Universal Robots PolyScope program: mt_rtde_control_loop_v4.urp

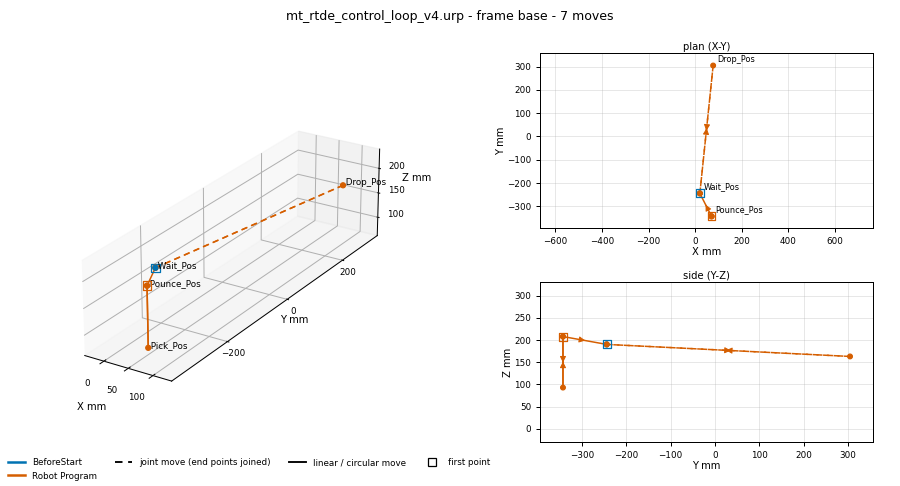
[picture p0: tool path of mt_rtde_control_loop_v4.urp in frame base, 7 of 7 moves have a stored position in this frame; points joined in program order, loops and branches not executed]
Program mt_rtde_control_loop_v4 (installation=mt_exhibit_v4 directory=/programs/usbdisk createdIn=3.2.19275.0 lastSavedIn=5.11.9.1010452 robotSerialNumber=20225300174)
Calibrated DH parameters: a=[-0.000135, -0.229339, -0.213305, 0.000029, -0.000076, 0]; d=[0.152122, 26.260282, -25.005713, -1.123774, 0.085381, 0.092263]; alpha=[1.57245, 0.003146, 0.006488, 1.570884, -1.571468, 0]; deltaTheta=[0, 0.345729, -0.307593, -0.038131, 0.000003, 0]
BeforeStart
  PRINTER_IDLE := 1
  PRINTER_RUNNING := 2
  COBOT_INIT := 0
  COBOT_IDLE := 1
  COBOT_PICKING := 2
  URCap Gripper Activate (Robotiq_Grippers, Robotiq Inc.) dataModel(ResetAndActivateKey=false)
  MoveJ speed 60 deg/s, acceleration 80 deg/s^2 (useActiveTCP=true) feature=mt_reference
    Waypoint Wait_Pos: TCP in base x=20.338 y=-244.22 z=190.23 mm, rx=-2.8747 ry=-1.2308 rz=0.0465 rad; joints [-50.864, -70.012, -95.058, -106.133, 88.723, -547.452] deg; TCP offset x=0 y=0 z=152.4 mm, rx=0 ry=0 rz=0 rad; feature pose in base x=182.345 y=-173.857 z=92.906 mm, rx=0.0004 ry=-0.0001 rz=-2.3564 rad
  SuppressedNode
    Set DigitalOutput pin=tool_out[0]; digitalValue=0
  URCap Gripper (Robotiq_Grippers, Robotiq Inc.) dataModel(position=0.0, force=100.0, speed=100.0, positionInDouble=0.0, forceInDouble=100.0, speedInDouble=100.0, slaveIds=[9], blocking=true)
  Script: rtde_set_watchdog("input_int_register_0", 1, "PAUSE")
  Script: write_output_integer_register(0, COBOT_INIT)
Robot Program (runOnlyOnce=false)
  Wait Condition expression=read_input_integer_register(0)≟PRINTER_IDLE
  'Ready to remove item from print bed'
  Script: write_output_integer_register(0,COBOT_PICKING)
  Folder Pick and Deposit
    MoveL speed 250 mm/s, acceleration 1200 mm/s^2 (useActiveTCP=true) feature=mt_reference
      Waypoint Pounce_Pos: TCP in base x=70.45 y=-342.866 z=207.922 mm, rx=2.8891 ry=1.2336 rz=0.0006 rad; joints [-56.166, -98.04, -66.059, -105.848, 90.24, -552.695] deg
    'Make sure grabber is open'
    MoveL speed 250 mm/s, acceleration 1200 mm/s^2 (useActiveTCP=true) feature=mt_reference
      Waypoint Pick_Pos: TCP in base x=70.517 y=-342.85 z=92.889 mm, rx=2.889 ry=1.2336 rz=0.0007 rad; joints [-56.257, -97.863, -97.534, -74.545, 90.252, -552.586] deg
    'Close grabber'
    SuppressedNode
      Set DigitalOutput pin=tool_out[1]; digitalValue=1
    URCap Gripper (Robotiq_Grippers, Robotiq Inc.) dataModel(position=100.0, force=100.0, speed=100.0, positionInDouble=100.0, forceInDouble=100.0, speedInDouble=100.0, slaveIds=[9], blocking=true)
    Wait Sleep waitTime=0.25
    SetPayload (workpieceName=Payload)
    MoveL speed 250 mm/s, acceleration 1200 mm/s^2 (useActiveTCP=true) feature=mt_reference
      Waypoint Pounce_Pos: TCP in base x=70.45 y=-342.866 z=207.922 mm, rx=2.8891 ry=1.2336 rz=0.0006 rad; joints [-56.166, -98.04, -66.059, -105.848, 90.24, -552.695] deg
      Waypoint Wait_Pos: TCP in base x=20.338 y=-244.22 z=190.23 mm, rx=-2.8747 ry=-1.2308 rz=0.0465 rad; joints [-50.864, -70.012, -95.058, -106.133, 88.723, -547.452] deg
    MoveJ speed 60 deg/s, acceleration 80 deg/s^2 (useActiveTCP=true) feature=mt_reference
      Waypoint Drop_Pos: TCP in base x=77.393 y=304.411 z=163.084 mm, rx=1.4186 ry=2.7868 rz=-0.0335 rad; joints [100.552, -88.496, -87.879, -95.061, 90.301, -475.701] deg
    'Drop Item'
    SuppressedNode
      Set DigitalOutput pin=tool_out[0]; digitalValue=0
    URCap Gripper (Robotiq_Grippers, Robotiq Inc.) dataModel(position=0.0, force=100.0, speed=100.0, positionInDouble=0.0, forceInDouble=100.0, speedInDouble=100.0, slaveIds=[9], blocking=true)
    Wait Sleep waitTime=0.25
    SetPayload (workpieceName=Payload)
    MoveJ speed 60 deg/s, acceleration 80 deg/s^2 (useActiveTCP=true) feature=mt_reference
      Waypoint Wait_Pos: TCP in base x=20.338 y=-244.22 z=190.23 mm, rx=-2.8747 ry=-1.2308 rz=0.0465 rad; joints [-50.864, -70.012, -95.058, -106.133, 88.723, -547.452] deg
  'Confirm pick and drop was completed'
  Script: write_output_integer_register(0,COBOT_IDLE)
  'Wait Until Client Controller Acknowledges Confirmation'
  Wait Condition expression=read_input_integer_register(0)≟PRINTER_RUNNING
  Script: sync()
